INTERFACE IListOfBytes EXTENDS IReadOnlyListOfBytes

METHOD Clear
VAR_INPUT
	releaseMemory : BOOL := FALSE;
END_VAR
END_METHOD

METHOD Find : BOOL
VAR_INPUT
	value : BYTE;
END_VAR
VAR_OUTPUT
	index : DINT;
END_VAR
END_METHOD

METHOD LoadFromAddress
VAR_INPUT
	sourceDataAddress : POINTER TO BYTE;
	sourceDataSize : DINT;
	startIndex : DINT := 0;
END_VAR
END_METHOD

METHOD LoadFromVariable
VAR_INPUT
	sourceVariable : ANY;
	startIndex : DINT := 0;
END_VAR
END_METHOD

METHOD Remove
VAR_INPUT
	value : BYTE;
END_VAR
END_METHOD

METHOD RemoveAt
VAR_INPUT
	index : DINT;
	count : DINT := 1;
END_VAR
END_METHOD

METHOD Resize
VAR_INPUT
	newBytesCount : DINT;
END_VAR
END_METHOD

METHOD Set
VAR_INPUT
	index : DINT;
	value : BYTE;
END_VAR
END_METHOD

END_INTERFACE

(* stored: Version 1.1.0.1
   Itf IListOfBytes: Id {518eb55c-df07-0206-0227-e692a273d945}
   Method Clear: Id {243fdc07-7928-4ca7-a298-f89f02bbd736}
   Method Find: Id {9318d27c-43e1-42e9-a8bf-c3a8b3921d40}
   Method LoadFromAddress: Id {f1c6da5c-ced0-42ee-9f57-c45302a7ebcb}
   Method LoadFromVariable: Id {b3c42220-f6d9-4c15-b9b4-e89b6fac55f8}
   Method Remove: Id {eed9e02a-e972-481f-8ddf-d0d8fccc576a}
   Method RemoveAt: Id {5d545c6c-7499-43af-8e59-315db670ead5}
   Method Resize: Id {c4504f91-d8a1-4fc4-bf4f-18aa14caa2ad}
   Method Set: Id {267c54d8-2df6-0ce5-162c-03537dc39a04} *)
